// TIA Portal V18 export
ORGANIZATION_BLOCK "Cyclic interrupt_axis_30ms"   // OB31, LAD, CyclicInterrupt
{ S7_Optimized_Access := 'TRUE' }
VERSION : 0.1
// stored: AutoNumber true, IsIECCheckEnabled false, SetENOAutomatically false
   VAR_INPUT
      Initial_Call : Bool;
      Event_Count : Int;
   END_VAR
BEGIN

REGION Network 1
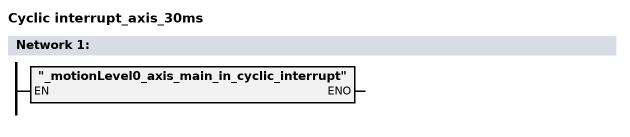
   RUNG wire#powerrail
      "_motionLevel0_axis_main_in_cyclic_interrupt"()
   END_RUNG
   // the same network as SCL:
   "_motionLevel0_axis_main_in_cyclic_interrupt"();
END_REGION
END_ORGANIZATION_BLOCK
